// TIA Portal V16 export
// export: Created 2021-07-12T14:47:19.8594162Z, ExportSetting WithDefaults, DisplayName Totally Integrated Automation Portal, DisplayVersion V16, DisplayName TIA Portal Version Control Interface, DisplayVersion V16, DisplayName TIA Portal Openness, DisplayVersion V16, DisplayName STEP 7 Professional, DisplayVersion V16, DisplayName STEP 7 Safety, DisplayVersion V16, DisplayName WinCC Professional, DisplayVersion V16
TYPE "LSimaHydTO_typeMeasurementConfig"
TITLE = LSimaHydTO_typeMeasurementConfig
// Configuration of the measurement function
// stored: IsFailsafeCompliant false
   STRUCT
      waitTimeMeasurement { S7_SetPoint := 'True'} : DInt := 100;   // Waiting time after ramping [ms]
      maxMeasurementTime { S7_SetPoint := 'True'} : DInt := 200;   // Measurement time [ms]
      offset { S7_SetPoint := 'True'} : LReal;   // Manipulated variable as drift compensation [%]
      safetyDistance { S7_SetPoint := 'True'} : LReal;   // Safety distance to avoid passing over the min. and max. positions
      forward { S7_SetPoint := 'True'} : "LSimaHydTO_typeMeasurementQOutput";   // Structure to define the manipulated variable
      backward { S7_SetPoint := 'True'} : "LSimaHydTO_typeMeasurementQOutput";   // Structure to define the manipulated variable
      numberOfRetryMeasurement { S7_SetPoint := 'True'} : Int := 1;   // Number of repeat attempts to measure the velocity, this parameter should be greater than / equal to 1
   END_STRUCT;
END_TYPE
